PROGRAM MAIN
VAR
	my_counter : INT := 0;
END_VAR

my_counter := my_counter + 1;

END_PROGRAM

(* stored: Version 1.1.0.1, ProductVersion 3.1.4024.12
   POU MAIN: Id {30cfc5af-b74e-445a-b332-297f92c143cd}, SpecialFunc None *)
